// TIA Portal V20 export
DATA_BLOCK "HmiInterface"   // DB97
{ DB_Accessible_From_OPC_UA := 'FALSE' }
AUTHOR : ERsystem_FA2_DH. Kim
// stored: Access Published, DBAccessibleFromOPCUA false, DBAccessibleFromWebserver false, MemoryReserve 100, Namespace Unit1.Em2
   VAR
      em : "LAF_typeEmInterface";
      cm : Struct
         null : Bool;
      END_STRUCT;
      semiAutoSplice : Struct
         jobs { S7_SetPoint := 'True'} : "LAF_typeJobsInterface";
         sequence { S7_SetPoint := 'True'} : "LAF_typeSequenceInterface";
      END_STRUCT;
      auxiliary : Struct
         parameters : Struct
            null : Bool;
         END_STRUCT;
         commands : Struct
            semiAutoSplicing1Times : Bool;
         END_STRUCT;
         monitoring : Struct
            null : Bool;
         END_STRUCT;
      END_STRUCT;
      cmSuctionPadTopUpDown : "LBC_typeTwoWayActuatorInterface";
      cmSuctionPadBtmUpDown { S7_SetPoint := 'True'} : "LBC_typeTwoWayActuatorInterface";
      cmCutterUpDown { S7_SetPoint := 'True'} : "LBC_typeTwoWayActuatorInterface";
      cmTapeTopUpDown { S7_SetPoint := 'True'} : "LBC_typeTwoWayActuatorInterface";
      cmTapeBtmUpDown { S7_SetPoint := 'True'} : "LBC_typeTwoWayActuatorInterface";
      cmSpliceHeadRotateTopFwdBwd { S7_SetPoint := 'True'} : "LBC_typeTwoWayActuatorInterface";
      cmSpliceHeadRotateBtmFwdBwd { S7_SetPoint := 'True'} : "LBC_typeTwoWayActuatorInterface";
      cmSuctionPadTopLeftVaccum { S7_SetPoint := 'True'} : "LBC_typeTwoWayActuatorInterface";
      cmSuctionPadTopRightVaccum { S7_SetPoint := 'True'} : "LBC_typeTwoWayActuatorInterface";
      cmSuctionPadBtmLeftVaccum { S7_SetPoint := 'True'} : "LBC_typeTwoWayActuatorInterface";
      cmSuctionPadBtmRightVaccum { S7_SetPoint := 'True'} : "LBC_typeTwoWayActuatorInterface";
      cmSuctionPadTopTapeVaccum { S7_SetPoint := 'True'} : "LBC_typeTwoWayActuatorInterface";
      cmSuctionPadBtmTapeVaccum { S7_SetPoint := 'True'} : "LBC_typeTwoWayActuatorInterface";
      intCondition : Struct
         Actuator_03 { S7_SetPoint := 'True'} : "LER.typeAxisActuatorCondition";   // SuctionPadTopUpDown
         Actuator_04 { S7_SetPoint := 'True'} : "LER.typeAxisActuatorCondition";   // SuctionPadBtmUpDown
         Actuator_05 { S7_SetPoint := 'True'} : "LER.typeAxisActuatorCondition";   // CutterUpDown
         Actuator_06 { S7_SetPoint := 'True'} : "LER.typeAxisActuatorCondition";   // TapeTopUpDown
         Actuator_07 { S7_SetPoint := 'True'} : "LER.typeAxisActuatorCondition";   // TapeBtmUpDown
         Actuator_08 { S7_SetPoint := 'True'} : "LER.typeAxisActuatorCondition";   // SpliceHeadRotateTopFwdBwd
         Actuator_09 { S7_SetPoint := 'True'} : "LER.typeAxisActuatorCondition";   // SpliceHeadRotateBtmFwdBwd
      END_STRUCT;
   END_VAR
BEGIN
END_DATA_BLOCK
